	{attribute 'TcLinkTo' := '.bLimitForwardEnable:=TIIB[EL7041-1000_XRTM1_Ydwn]^STM Status^Status^Digital input 1;
                              .bLimitBackwardEnable:=TIIB[EL7041-1000_XRTM1_Ydwn]^STM Status^Status^Digital input 2'}
	{attribute 'pytmc' := '
		pv: XRTMR1:HOMS:MMS:YDWN
	'}
	M2 : DUT_MotionStage := (fVelocity:=200.0, nEnableMode:=ENUM_StageEnableMode.ALWAYS, bPowerSelf:=TRUE); // XRTM1 Ydwn
	fbMotionStage_m2 : FB_MotionStage;

	{attribute 'TcLinkTo' := '.bLimitForwardEnable:=TIIB[EL7041-1000_XRTM1_Xup]^STM Status^Status^Digital input 1;
                              .bLimitBackwardEnable:=TIIB[EL7041-1000_XRTM1_Xup]^STM Status^Status^Digital input 2'}
	{attribute 'pytmc' := '
		pv: XRTMR1:HOMS:MMS:XUP
	'}
	M3 : DUT_MotionStage := (fVelocity:=1000.0, nEnableMode:=ENUM_StageEnableMode.ALWAYS, bPowerSelf:=TRUE); // XRTM1 Xup
	fbMotionStage_m3 : FB_MotionStage;

	{attribute 'TcLinkTo' := '.bLimitForwardEnable:=TIIB[EL7041-1000_XRTM1_Xdwn]^STM Status^Status^Digital input 1;
                              .bLimitBackwardEnable:=TIIB[EL7041-1000_XRTM1_Xdwn]^STM Status^Status^Digital input 2'}
	{attribute 'pytmc' := '
		pv: XRTMR1:HOMS:MMS:XDWN
	'}
	M4 : DUT_MotionStage := (fVelocity:=1000.0, nEnableMode:=ENUM_StageEnableMode.ALWAYS, bPowerSelf:=TRUE); // XRTM1 Xdwn
	fbMotionStage_m4 : FB_MotionStage;

	{attribute 'TcLinkTo' := '.bLimitForwardEnable:=TIIB[EL7041-1000_XRTM1_PitchCoarse]^STM Status^Status^Digital input 1;
                              .bLimitBackwardEnable:=TIIB[EL7041-1000_XRTM1_PitchCoarse]^STM Status^Status^Digital input 2'}
	{attribute 'pytmc' := '
		pv: XRTMR1:HOMS:MMS:PITCH
	'}
	M5 : DUT_MotionStage := (fVelocity:=150.0); // XRTM1 Pitch Stepper

	{attribute 'TcLinkTo' := '.bLimitForwardEnable:=TIIB[EL7041-1000_XRTM1_Bender]^STM Status^Status^Digital input 1;
                              .bLimitBackwardEnable:=TIIB[EL7041-1000_XRTM1_Bender]^STM Status^Status^Digital input 2'}
	{attribute 'pytmc' := '
		pv: XRTMR1:HOMS:MMS:BENDER
	'}
	M6 : DUT_MotionStage := (fVelocity:=150.0, nEnableMode:=ENUM_StageEnableMode.ALWAYS, bPowerSelf:=TRUE); // XRTM1 Bender
	fbMotionStage_m6 : FB_MotionStage;

	{attribute 'TcLinkTo' := '.fbRunHOMS.bSTOEnable1:=TIIB[EL1004_XRTM1_STO]^Channel 1^Input;
                              .fbRunHOMS.bSTOEnable2:=TIIB[EL1004_XRTM1_STO]^Channel 2^Input;
	                          .fbRunHOMS.stYupEnc.Count:=TIIB[EL5042_XRTM1_Yupdwn]^FB Inputs Channel 1^Position;
	                          .fbRunHOMS.stYdwnEnc.Count:=TIIB[EL5042_XRTM1_Yupdwn]^FB Inputs Channel 2^Position;
	                          .fbRunHOMS.stXupEnc.Count:=TIIB[EL5042_XRTM1_Xupdwn]^FB Inputs Channel 1^Position;
	                          .fbRunHOMS.stXdwnEnc.Count:=TIIB[EL5042_XRTM1_Xupdwn]^FB Inputs Channel 2^Position'}
	{attribute 'pytmc' := '
		pv: XRTMR1:HOMS
	'}
	XRTM1 : DUT_HOMS;

	// Encoder Arrays/RMS Watch:
	{attribute 'pytmc' := '
		pv: XRTMR1:HOMS:ENC:Y
	'}
	fbYRMSErrorXRTM1 : FB_RMSWatch;
	fMaxYRMSErrorXRTM1 : LREAL;
	fMinYRMSErrorXRTM1 : LREAL;

	{attribute 'pytmc' := '
		pv: XRTMR1:HOMS:ENC:X
	'}
	fbXRMSErrorXRTM1 : FB_RMSWatch;
	fMaxXRMSErrorXRTM1 : LREAL;
	fMinXRMSErrorXRTM1 : LREAL;

	{attribute 'pytmc' := '
		pv: XRTMR1:HOMS:ENC:PITCH
	'}
	fbPitchRMSErrorXRTM1 : FB_RMSWatch;
	fMaxPitchRMSErrorXRTM1 : LREAL;
	fMinPitchRMSErrorXRTM1 : LREAL;

	{attribute 'pytmc' := '
		pv: XRTMR1:HOMS:ENC:BENDER
	'}
	fbBenderRMSErrorXRTM1 : FB_RMSWatch;
	fMaxBenderRMSErrorXRTM1 : LREAL;
	fMinBenderRMSErrorXRTM1 : LREAL;

	// Pitch Control
	fbXRTM1PitchControl : FB_PitchControl;
	bXRTM1PitchDone : BOOL;
	bXRTM1PitchBusy : BOOL;

	// Bender Control
	fbBenderXRTM1 : FB_Bender;

	// Raw Encoder Counts
	{attribute 'pytmc' := '
		pv: XRTMR1:HOMS:ENC:YUP:CNT
		field: EGU cnt
		io: i
	'}
	nEncCntYupXRTM1 : UDINT;
	{attribute 'pytmc' := '
		pv: XRTMR1:HOMS:ENC:YDWN:CNT
		field: EGU cnt
		io: i
	'}
	nEncCntYdwnXRTM1 : UDINT;
	{attribute 'pytmc' := '
		pv: XRTMR1:HOMS:ENC:XUP:CNT
		field: EGU cnt
		io: i
	'}
	nEncCntXupXRTM1 : UDINT;
	{attribute 'pytmc' := '
		pv: XRTMR1:HOMS:ENC:XDWN:CNT
		field: EGU cnt
		io: i
	'}
	nEncCntXdwnXRTM1 : UDINT;
	{attribute 'pytmc' := '
		pv: XRTMR1:HOMS:ENC:PITCH:CNT
		field: EGU cnt
		io: i
	'}
	nEncCntPitchXRTM1 : UDINT;

	// Encoder Reference Values
	{attribute 'pytmc' := '
		pv: XRTMR1:HOMS:ENC:YUP:REF
		field: EGU cnt
		io: i
	'}
	nEncRefYupXRTM1 : UDINT;
	{attribute 'pytmc' := '
		pv: XRTMR1:HOMS:ENC:YDWN:REF
		field: EGU cnt
		io: i
	'}
	nEncRefYdwnXRTM1 : UDINT;
	{attribute 'pytmc' := '
		pv: XRTMR1:HOMS:ENC:XUP:REF
		field: EGU cnt
		io: i
	'}
	nEncRefXupXRTM1 : UDINT;
	{attribute 'pytmc' := '
		pv: XRTMR1:HOMS:ENC:XDWN:REF
		field: EGU cnt
		io: i
	'}
	nEncRefXdwnXRTM1 : UDINT;
	{attribute 'pytmc' := '
		pv: XRTMR1:HOMS:ENC:PITCH:REF
		field: EGU cnt
		io: i
	'}
	nEncRefPitchXRTM1 : UDINT;
	mcReadParameterPitchXRTM1 : MC_ReadParameter;
	fEncRefPitchXRTM1_urad : LREAL; // Current Pitch encoder offset in urad
	
    //****** HOMS M2 and M3 **************************
	tpImAPLC : TP := (PT:=T#10S);
	ExpertMode	:	BOOL := FALSE;
	PitchManualMode: BOOL := FALSE;
	
	//Drive CoE Fb
	fbY1CoE	:	FB_ElmoGDCBellCoE;
	fbY2CoE	:	FB_ElmoGDCBellCoE;
	
	fbX1CoE	:	FB_ElmoGDCBellCoE;
	fbX2CoE	:	FB_ElmoGDCBellCoE;
	
	fbP1CoE	:	FB_ElmoGDCBellCoE;
	fbB1CoE	:	FB_ElmoGDCBellCoE;
	
	//Init params trigger
	rtInitParams	:	R_TRIG;
	
	//Test Parameters
	rStepSize: REAL;
	SettleTime: TON := (
	PT:=T#2s);
	TestUpperVoltage: REAL := 100;
	TestLowerVoltage: REAL := 10;
	xRunPiezoRepeatTest: BOOL;
	
	//Drive reference initializations
	fbInitDriveRef	:	FB_InitDriveRefs;
	//MPS Information
	fbMPS_States :  FB_MPS_STATES;
	M2_INRANGE  :   ARRAY[0..1] OF DINT := [24568920, 26568920];
	M2_OUTRANGE  :  ARRAY[0..1] OF DINT := [43568250, 50570250];
	//noConsequence	:	BOOL;
	
	mcBenderPower	:	MC_POWER;
	
	// HOMS M2
	XRTM2PitchControl	    :	FB_PitchControlOld;
	XRTM2Y_GantryControl	:	FB_Gantry;
	XRTM2X_GantryControl	:	FB_Gantry;
	
	fbM2Y1LS	:	FB_LimitSwitchState;
	fbM2Y2LS	:	FB_LimitSwitchState;
	fbM2X1LS	:	FB_LimitSwitchState;
	fbM2X2LS	:	FB_LimitSwitchState;
	fbM2P1LS	:	FB_PitchSoftLimits;	
	
    // HOMS M3
	XRTM3PitchControl	    :	FB_PitchControlOld;
	XRTM3Y_GantryControl	:	FB_Gantry;
	XRTM3X_GantryControl	:	FB_Gantry;
	
	fbM3Y1LS	:	FB_LimitSwitchState;
	fbM3Y2LS	:	FB_LimitSwitchState;
	fbM3X1LS	:	FB_LimitSwitchState;
	fbM3X2LS	:	FB_LimitSwitchState;
	fbM3P1LS	:	FB_PitchSoftLimits;	
	
	//************** **** *** ** *
	
	
	
	// PMPS arbiter interface
	fbArbiterIO : FB_SubSysToArbiter_IO;
	
	// Common
	fEncLeverArm_mm : LREAL := 513.0;
	// Logging
	fbLogHandler : FB_LogHandler;

END_VAR

// XRTM1
XRTM1.fbRunHOMS(stYup:=M1,
               stYdwn:=M2,
               stXup:=M3,
               stXdwn:=M4,
               stPitch:=M5,
	           nYupEncRef:=GVL_XRTM1_Constants.nYUP_ENC_REF,
               nYdwnEncRef:=GVL_XRTM1_Constants.nYDWN_ENC_REF,
               nXupEncRef:=GVL_XRTM1_Constants.nXUP_ENC_REF,
               nXdwnEncRef:=GVL_XRTM1_Constants.nXDWN_ENC_REF,
			   bExecuteCoupleY:=XRTM1.bExecuteCoupleY,
               bExecuteCoupleX:=XRTM1.bExecuteCoupleX,
			   bExecuteDecoupleY:=XRTM1.bExecuteDecoupleY,
               bExecuteDecoupleX:=XRTM1.bExecuteDecoupleX,
               bGantryAlreadyCoupledY=>XRTM1.bGantryAlreadyCoupledY,
               bGantryAlreadyCoupledX=>XRTM1.bGantryAlreadyCoupledX,
               nCurrGantryY=>XRTM1.nCurrGantryY,
               nCurrGantryX=>XRTM1.nCurrGantryX);
fbBenderXRTM1(stBender:=M6,
	         bSTOEnable1:=XRTM1.fbRunHOMS.bSTOEnable1,
		     bSTOEnable2:=XRTM1.fbRunHOMS.bSTOEnable2);
// No slave motion through Epics
M2.bExecute := FALSE; // XRTM1-Ydwn
M4.bExecute := FALSE; // XRTM1-Xdwn

// Convert nCurrGantry to um (smaller number) to read out in epics
XRTM1.fCurrGantryY_um := LINT_TO_REAL(XRTM1.nCurrGantryY) / 1000.0;
XRTM1.fCurrGantryX_um := LINT_TO_REAL(XRTM1.nCurrGantryX) / 1000.0;

// FB_MotionStage's for non-piezo axes
fbMotionStage_m1(stMotionStage:=M1);
fbMotionStage_m2(stMotionStage:=M2);
fbMotionStage_m3(stMotionStage:=M3);
fbMotionStage_m4(stMotionStage:=M4);
fbMotionStage_m6(stMotionStage:=M6);

// Calculate Pitch RMS Error:
fbYRMSErrorXRTM1(stMotionStage:=M1,
	            fMaxRMSError=>fMaxYRMSErrorXRTM1,
				fMinRMSError=>fMinYRMSErrorXRTM1);

fbXRMSErrorXRTM1(stMotionStage:=M3,
	            fMaxRMSError=>fMaxXRMSErrorXRTM1,
				fMinRMSError=>fMinXRMSErrorXRTM1);

fbPitchRMSErrorXRTM1(stMotionStage:=M5,
	                fMaxRMSError=>fMaxPitchRMSErrorXRTM1,
					fMinRMSError=>fMinPitchRMSErrorXRTM1);

fbBenderRMSErrorXRTM1(stMotionStage:=M6,
	                 fMaxRMSError=>fMaxBenderRMSErrorXRTM1,
					 fMinRMSError=>fMinBenderRMSErrorXRTM1);
// Pitch Control
fbXRTM1PitchControl(Pitch:=GVL_XRTM1.XRTM1_Pitch,
				   Stepper:=M5,
				   lrCurrentSetpoint:=M5.fPosition,
                   q_bDone=>bXRTM1PitchDone,
                   q_bBusy=>bXRTM1PitchBusy);
// When STO hit, need to reset SP
IF NOT M5.bHardwareEnable THEN
	M5.fPosition := M5.stAxisStatus.fActPosition;
END_IF

// Raw Encoder Counts For Epics
nEncCntYupXRTM1 := ULINT_TO_UDINT(XRTM1.fbRunHOMS.stYupEnc.Count);
nEncCntYdwnXRTM1 := ULINT_TO_UDINT(XRTM1.fbRunHOMS.stYdwnEnc.Count);
nEncCntXupXRTM1 := ULINT_TO_UDINT(XRTM1.fbRunHOMS.stXupEnc.Count);
nEncCntXdwnXRTM1 := ULINT_TO_UDINT(XRTM1.fbRunHOMS.stXdwnEnc.Count);
nEncCntPitchXRTM1 := LINT_TO_UDINT(GVL_XRTM1.XRTM1_Pitch.diEncCnt);

// Encoder Reference Values For Epics
nEncRefYupXRTM1 := ULINT_TO_UDINT(GVL_XRTM1_Constants.nYUP_ENC_REF);
nEncRefYdwnXRTM1 := ULINT_TO_UDINT(GVL_XRTM1_Constants.nYDWN_ENC_REF);
nEncRefXupXRTM1 := ULINT_TO_UDINT(GVL_XRTM1_Constants.nXUP_ENC_REF);
nEncRefXdwnXRTM1 := ULINT_TO_UDINT(GVL_XRTM1_Constants.nXDWN_ENC_REF);
mcReadParameterPitchXRTM1(Axis:=M5.Axis,
	                     Enable:=TRUE,
				         ParameterNumber:=MC_AxisParameter.AxisEncoderOffset,
				         ReadMode:=READMODE_CYCLIC,
				         Value=>fEncRefPitchXRTM1_urad);

nEncRefPitchXRTM1 := LREAL_TO_UDINT(ABS(fEncRefPitchXRTM1_urad) * fEncLeverArm_mm);

// HOMS ************************ ***** **** *** ** *
p_ModbusRx_OutputCoils();
p_ModbusRx_PLCMemory();

//InitParams
////////////////////
rtInitParams(CLK:=gFirstPass);
IF rtInitParams.Q THEN
	Init_XRTM2();
	Init_XRTM3();
	gFirstPass := FALSE;
END_IF

//System Error Handling
/////////////////////////////////////
//SystemErrorSummary(); //Check this action for a summary of all system faults
					  
//SystemError();

//Driver Parameter Verification
/////////////////////////////////////

//Gantry Interlock Logic
/////////////////////////////////////
	//SimGantry.VAxis.i_xMotorInterlock := TRUE;
	//SimGantry.PAxis.i_xMotorInterlock := TRUE;
	//SimGantry.SAxis.i_xMotorInterlock := TRUE;
	
LimitSwitchIO();

// Pitch control
/////////////////////////////////////
XRTM2PitchControl(Pitch:=HOMS2_Pitch, DirectPiezoMode:=(ExpertMode AND PitchManualMode), q_xDone=>HOMS2_Pitch.Axis.bDone, q_xBusy => HOMS2_Pitch.Axis.bBusy);
XRTM3PitchControl(Pitch:=HOMS3_Pitch, DirectPiezoMode:=(ExpertMode AND PitchManualMode), q_xDone=>HOMS3_Pitch.Axis.bDone, q_xBusy => HOMS3_Pitch.Axis.bBusy);
//Y motion
/////////////////////////////////////
HOMS3_YGantry.PAxis.stAxis.ReadStatus();
HOMS3_YGantry.SAxis.stAxis.ReadStatus();
HOMS3_YGantry.PAxis.stStatus.rActPosition := LREAL_TO_REAL(HOMS3_YGantry.PAxis.stAxis.NcToPlc.ActPos);
HOMS3_YGantry.SAxis.stStatus.rActPosition := LREAL_TO_REAL(HOMS3_YGantry.SAxis.stAxis.NcToPlc.ActPos);

//X Motion
/////////////////////////////////////
XRTM2X_GantryControl(Gantry:=HOMS2_XGantry);
XRTM3X_GantryControl(Gantry:=HOMS3_XGantry);

//Communicate state to MPS
////////////////////////////////
fbMPS_States(GANTRY:=HOMS2_XGantry,
			 OUT_LS:=NOT HOMS2_XGantry.PAxis.xHiLS OR NOT HOMS2_XGantry.SAxis.xLoLS,
			 IN_RANGE:=M2_INRANGE,
			 OUT_RANGE:=M2_OUTRANGE);
			 
bXRT_M2_IN  := fbMPS_States.IN;
bXRT_M2_OUT := fbMPS_States.OUT;
//EPICS Tx Update
////////////////////
p_ModbusTx_InputCoils();
//p_ModbusTx_OutputCoils();
p_ModbusTx_InputReg();
p_ModbusTx_PLCMemory();

// **************************** ***** **** *** ** * HOMS


P_CoatingProtections();

// Logging
fbLogHandler();

// PMPS
GVL_PMPS.g_fbArbiter1.AddRequest(16#5, PMPS_GVL.cstFullBeam);
fbArbiterIO(Arbiter := GVL_PMPS.g_fbArbiter1, fbFFHWO := GVL_PMPS.g_FastFaultOutput1);
GVL_PMPS.g_FastFaultOutput1.Execute(i_xVeto:=);
GVL_PMPS.g_FastFaultOutput2.Execute(i_xVeto:=);

ACTION Init_XRTM2:
//FEE-M2
///////////////////////////


//Initialize ELMO Drive references
fbInitDriveRef(stCoE:=HOMS2_XGantry.PAxis.stCoE);
fbInitDriveRef(stCoE:=HOMS2_XGantry.SAxis.stCoE);
fbInitDriveRef(stCoE:=HOMS2_YGantry.PAxis.stCoE);
fbInitDriveRef(stCoE:=HOMS2_YGantry.SAxis.stCoE);
fbInitDriveRef(stCoE:=HOMS2_Pitch.Stepper.stCoE);

//Initialze Drive Speeds and Accelerations
//////////////////////////////////////////
HOMS2_XGantry.PAxis.fAcceleration := 1.0;
HOMS2_XGantry.SAxis.fAcceleration := 1.0;
HOMS2_YGantry.PAxis.fAcceleration := 1.0;
HOMS2_YGantry.SAxis.fAcceleration := 1.0;

HOMS2_XGantry.PAxis.fDeceleration := 1.0;
HOMS2_XGantry.SAxis.fDeceleration := 1.0;
HOMS2_YGantry.PAxis.fDeceleration := 1.0;
HOMS2_YGantry.SAxis.fDeceleration := 1.0;

HOMS2_XGantry.PAxis.fVelocity := 0.1;
HOMS2_XGantry.SAxis.fVelocity := 0.1;
HOMS2_YGantry.PAxis.fVelocity := 0.1;
HOMS2_YGantry.SAxis.fVelocity := 0.1;

HOMS2_Pitch.Stepper.fAcceleration := 39;
HOMS2_Pitch.Stepper.fDeceleration := 39;
HOMS2_Pitch.Stepper.fVelocity     := 100;

//Initialize Piezo Driver
/////////////////////////////////////
HOMS2_Pitch.Piezo.stPIParams.fKp := 0.001;
HOMS2_Pitch.Piezo.stPIParams.tTn := T#500MS;
HOMS2_Pitch.Piezo.stPIParams.fOutMaxLimit := 1;
HOMS2_Pitch.Piezo.stPIParams.fOutMinLimit := -1;
END_ACTION

ACTION Init_XRTM3:
//FEE-M3
///////////////////////////


//Initialize ELMO Drive references
fbInitDriveRef(stCoE:=HOMS3_XGantry.PAxis.stCoE);
fbInitDriveRef(stCoE:=HOMS3_XGantry.SAxis.stCoE);
fbInitDriveRef(stCoE:=HOMS3_YGantry.PAxis.stCoE);
fbInitDriveRef(stCoE:=HOMS3_YGantry.SAxis.stCoE);
fbInitDriveRef(stCoE:=HOMS3_Pitch.Stepper.stCoE);

//Initialze Drive Speeds and Accelerations
//////////////////////////////////////////
HOMS3_XGantry.PAxis.fAcceleration := 1.0;
HOMS3_XGantry.SAxis.fAcceleration := 1.0;
HOMS3_YGantry.PAxis.fAcceleration := 1.0;
HOMS3_YGantry.SAxis.fAcceleration := 1.0;

HOMS3_XGantry.PAxis.fDeceleration := 1.0;
HOMS3_XGantry.SAxis.fDeceleration := 1.0;
HOMS3_YGantry.PAxis.fDeceleration := 1.0;
HOMS3_YGantry.SAxis.fDeceleration := 1.0;

HOMS3_XGantry.PAxis.fVelocity := 0.1;
HOMS3_XGantry.SAxis.fVelocity := 0.1;
HOMS3_YGantry.PAxis.fVelocity := 0.1;
HOMS3_YGantry.SAxis.fVelocity := 0.1;

HOMS3_Pitch.Stepper.fAcceleration := 39;
HOMS3_Pitch.Stepper.fDeceleration := 39;
HOMS3_Pitch.Stepper.fVelocity     := 100;

//Initialize Piezo Driver
/////////////////////////////////////
HOMS3_Pitch.Piezo.stPIParams.fKp := 0.001;
HOMS3_Pitch.Piezo.stPIParams.tTn := T#500MS;
HOMS3_Pitch.Piezo.stPIParams.fOutMaxLimit := 1;
HOMS3_Pitch.Piezo.stPIParams.fOutMinLimit := -1;
END_ACTION

ACTION LimitSwitchIO:
//XRT M2
//////////////////////////
fbM2Y1LS(diInputs:=HOMS2_YGantry.PAxis.diInputs, 
xHiLS=>HOMS2_YGantry.PAxis.xHiLS,
xLoLS=>HOMS2_YGantry.PAxis.xLoLS,
STO => gM2STO);

fbM2Y2LS(diInputs:=HOMS2_YGantry.SAxis.diInputs, 
xHiLS=>HOMS2_YGantry.SAxis.xHiLS,
xLoLS=>HOMS2_YGantry.SAxis.xLoLS);

fbM2X1LS(diInputs:=HOMS2_XGantry.PAxis.diInputs, 
xHiLS=>HOMS2_XGantry.PAxis.xHiLS,
xLoLS=>HOMS2_XGantry.PAxis.xLoLS);

fbM2X2LS(diInputs:=HOMS2_XGantry.SAxis.diInputs, 
xHiLS=>HOMS2_XGantry.SAxis.xHiLS,
xLoLS=>HOMS2_XGantry.SAxis.xLoLS);

fbM2P1LS(Pitch:=HOMS2_Pitch,
xHiLS=>HOMS2_Pitch.Stepper.xHiLS,
xLoLS=>HOMS2_Pitch.Stepper.xLoLS);

//XRT M3
//////////////////////////
fbM3Y1LS(diInputs:=HOMS3_YGantry.PAxis.diInputs, 
xHiLS=>HOMS3_YGantry.PAxis.xHiLS,
xLoLS=>HOMS3_YGantry.PAxis.xLoLS,
STO => gM3STO);

fbM3Y2LS(diInputs:=HOMS3_YGantry.SAxis.diInputs, 
xHiLS=>HOMS3_YGantry.SAxis.xHiLS,
xLoLS=>HOMS3_YGantry.SAxis.xLoLS);

fbM3X1LS(diInputs:=HOMS3_XGantry.PAxis.diInputs, 
xHiLS=>HOMS3_XGantry.PAxis.xHiLS,
xLoLS=>HOMS3_XGantry.PAxis.xLoLS);
(*
fbM3X2LS(diInputs:=HOMS3_XGantry.PAxis.diInputs,  //Paxis is here on purpose <HACK>
xHiLS=>HOMS3_XGantry.SAxis.xHiLS,
xLoLS=>HOMS3_XGantry.SAxis.xLoLS);
*)
fbM3X2LS(diInputs:=HOMS3_XGantry.SAxis.diInputs,  // Switching to SAxis works as expected, reason for <HACK> unclear
xHiLS=>HOMS3_XGantry.SAxis.xHiLS,
xLoLS=>HOMS3_XGantry.SAxis.xLoLS);

fbM3P1LS(Pitch:=HOMS3_Pitch,
xHiLS=>HOMS3_Pitch.Stepper.xHiLS,
xLoLS=>HOMS3_Pitch.Stepper.xLoLS);
END_ACTION

END_PROGRAM

// ---- POUs/Modbus/p_ModbusRx_OutputCoils.TcPOU
PROGRAM p_ModbusRx_OutputCoils
VAR
	
END_VAR

HOMS2_XGantry.PAxis.bTwkFwd:=mb_Output_Coils[60];
HOMS2_XGantry.PAxis.bTwkBwd:=mb_Output_Coils[61];
HOMS2_XGantry.SAxis.bTwkFwd:=mb_Output_Coils[62];
HOMS2_XGantry.SAxis.bTwkBwd:=mb_Output_Coils[63];
HOMS2_YGantry.PAxis.bTwkFwd:=mb_Output_Coils[64];
HOMS2_YGantry.PAxis.bTwkBwd:=mb_Output_Coils[65];
HOMS2_YGantry.SAxis.bTwkFwd:=mb_Output_Coils[66];
HOMS2_YGantry.SAxis.bTwkBwd:=mb_Output_Coils[67];
HOMS2_Pitch.Axis.bTwkFwd:=mb_Output_Coils[68];
HOMS2_Pitch.Axis.bTwkBwd:=mb_Output_Coils[69];
HOMS2_Pitch.Axis.xStop:=mb_Output_Coils[73];
HOMS2_XGantry.xUncouple:=mb_Output_Coils[76];
HOMS2_YGantry.xUncouple:=mb_Output_Coils[77];
HOMS3_XGantry.PAxis.bTwkFwd:=mb_Output_Coils[78];
HOMS3_XGantry.PAxis.bTwkBwd:=mb_Output_Coils[79];
HOMS3_XGantry.SAxis.bTwkFwd:=mb_Output_Coils[80];
HOMS3_XGantry.SAxis.bTwkBwd:=mb_Output_Coils[81];
HOMS3_YGantry.PAxis.bTwkFwd:=mb_Output_Coils[82];
HOMS3_YGantry.PAxis.bTwkBwd:=mb_Output_Coils[83];
HOMS3_YGantry.SAxis.bTwkFwd:=mb_Output_Coils[84];
HOMS3_YGantry.SAxis.bTwkBwd:=mb_Output_Coils[85];
HOMS3_Pitch.Axis.bTwkFwd:=mb_Output_Coils[86];
HOMS3_Pitch.Axis.bTwkBwd:=mb_Output_Coils[87];
HOMS3_Pitch.Piezo.xEnable:=mb_Output_Coils[88];
HOMS3_Pitch.Axis.xStop:=mb_Output_Coils[89];
HOMS3_XGantry.xUncouple:=mb_Output_Coils[90];
HOMS3_YGantry.xUncouple:=mb_Output_Coils[91];
HOMS2_XGantry.PAxis.xReset := mb_Output_Coils[95];
HOMS2_YGantry.PAxis.xReset := mb_Output_Coils[96];
HOMS2_Pitch.Axis.xReset := mb_Output_Coils[97];
HOMS3_XGantry.PAxis.xReset := mb_Output_Coils[98];
HOMS3_YGantry.PAxis.xReset := mb_Output_Coils[99];
HOMS3_Pitch.Axis.xReset := mb_Output_Coils[100];

END_PROGRAM

// ---- POUs/Modbus/p_ModbusRx_PLCMemory.TcPOU
PROGRAM p_ModbusRx_PLCMemory
VAR
END_VAR

MEMCPY(srcAddr:=ADR(mb_PLC_Memory[20]), destAddr:=ADR(HOMS2_XGantry.PAxis.rReqAbsolute), n:=SIZEOF(HOMS2_XGantry.PAxis.rReqAbsolute));
MEMCPY(srcAddr:=ADR(mb_PLC_Memory[22]), destAddr:=ADR(HOMS2_XGantry.PAxis.rTweak), n:=SIZEOF(HOMS2_XGantry.PAxis.rTweak));
MEMCPY(srcAddr:=ADR(mb_PLC_Memory[24]), destAddr:=ADR(HOMS2_XGantry.SAxis.rReqAbsolute), n:=SIZEOF(HOMS2_XGantry.SAxis.rReqAbsolute));
MEMCPY(srcAddr:=ADR(mb_PLC_Memory[26]), destAddr:=ADR(HOMS2_XGantry.SAxis.rTweak), n:=SIZEOF(HOMS2_XGantry.SAxis.rTweak));
MEMCPY(srcAddr:=ADR(mb_PLC_Memory[28]), destAddr:=ADR(HOMS2_YGantry.PAxis.rReqAbsolute), n:=SIZEOF(HOMS2_YGantry.PAxis.rReqAbsolute));
MEMCPY(srcAddr:=ADR(mb_PLC_Memory[30]), destAddr:=ADR(HOMS2_YGantry.PAxis.rTweak), n:=SIZEOF(HOMS2_YGantry.PAxis.rTweak));
MEMCPY(srcAddr:=ADR(mb_PLC_Memory[32]), destAddr:=ADR(HOMS2_YGantry.SAxis.rReqAbsolute), n:=SIZEOF(HOMS2_YGantry.SAxis.rReqAbsolute));
MEMCPY(srcAddr:=ADR(mb_PLC_Memory[34]), destAddr:=ADR(HOMS2_YGantry.SAxis.rTweak), n:=SIZEOF(HOMS2_YGantry.SAxis.rTweak));
MEMCPY(srcAddr:=ADR(mb_PLC_Memory[36]), destAddr:=ADR(HOMS2_Pitch.Axis.rReqAbsPos), n:=SIZEOF(HOMS2_Pitch.Axis.rReqAbsPos));
MEMCPY(srcAddr:=ADR(mb_PLC_Memory[38]), destAddr:=ADR(HOMS2_Pitch.Axis.rTweak), n:=SIZEOF(HOMS2_Pitch.Axis.rTweak));
MEMCPY(srcAddr:=ADR(mb_PLC_Memory[40]), destAddr:=ADR(HOMS3_XGantry.PAxis.rReqAbsolute), n:=SIZEOF(HOMS3_XGantry.PAxis.rReqAbsolute));
MEMCPY(srcAddr:=ADR(mb_PLC_Memory[42]), destAddr:=ADR(HOMS3_XGantry.PAxis.rTweak), n:=SIZEOF(HOMS3_XGantry.PAxis.rTweak));
MEMCPY(srcAddr:=ADR(mb_PLC_Memory[44]), destAddr:=ADR(HOMS3_XGantry.SAxis.rReqAbsolute), n:=SIZEOF(HOMS3_XGantry.SAxis.rReqAbsolute));
MEMCPY(srcAddr:=ADR(mb_PLC_Memory[46]), destAddr:=ADR(HOMS3_XGantry.SAxis.rTweak), n:=SIZEOF(HOMS3_XGantry.SAxis.rTweak));
MEMCPY(srcAddr:=ADR(mb_PLC_Memory[48]), destAddr:=ADR(HOMS3_YGantry.PAxis.rReqAbsolute), n:=SIZEOF(HOMS3_YGantry.PAxis.rReqAbsolute));
MEMCPY(srcAddr:=ADR(mb_PLC_Memory[50]), destAddr:=ADR(HOMS3_YGantry.PAxis.rTweak), n:=SIZEOF(HOMS3_YGantry.PAxis.rTweak));
MEMCPY(srcAddr:=ADR(mb_PLC_Memory[52]), destAddr:=ADR(HOMS3_YGantry.SAxis.rReqAbsolute), n:=SIZEOF(HOMS3_YGantry.SAxis.rReqAbsolute));
MEMCPY(srcAddr:=ADR(mb_PLC_Memory[54]), destAddr:=ADR(HOMS3_YGantry.SAxis.rTweak), n:=SIZEOF(HOMS3_YGantry.SAxis.rTweak));
MEMCPY(srcAddr:=ADR(mb_PLC_Memory[56]), destAddr:=ADR(HOMS3_Pitch.Axis.rReqAbsPos), n:=SIZEOF(HOMS3_Pitch.Axis.rReqAbsPos));
MEMCPY(srcAddr:=ADR(mb_PLC_Memory[58]), destAddr:=ADR(HOMS3_Pitch.Axis.rTweak), n:=SIZEOF(HOMS3_Pitch.Stepper.rTweak));

MEMCPY(srcAddr:=ADR(mb_PLC_Memory[64]), destAddr:=ADR(HOMS2_Pitch.Stepper.rStepperDmovRange), n:=SIZEOF(HOMS2_Pitch.Stepper.rStepperDmovRange));
MEMCPY(srcAddr:=ADR(mb_PLC_Memory[66]), destAddr:=ADR(HOMS2_Pitch.Piezo.rPiezoDmovRange), n:=SIZEOF(HOMS2_Pitch.Piezo.rPiezoDmovRange));
MEMCPY(srcAddr:=ADR(mb_PLC_Memory[68]), destAddr:=ADR(HOMS3_Pitch.Stepper.rStepperDmovRange), n:=SIZEOF(HOMS3_Pitch.Stepper.rStepperDmovRange));
MEMCPY(srcAddr:=ADR(mb_PLC_Memory[70]), destAddr:=ADR(HOMS3_Pitch.Piezo.rPiezoDmovRange), n:=SIZEOF(HOMS3_Pitch.Piezo.rPiezoDmovRange));

//MEMCPY(srcAddr:=ADR(mb_PLC_Memory[140]), destAddr:=ADR(HOMS1_Pitch.Piezo.rReqVoltage), n:=SIZEOF(HOMS1_Pitch.Piezo.rReqVoltage));
//MEMCPY(srcAddr:=ADR(mb_PLC_Memory[142]), destAddr:=ADR(HOMS2_Pitch.Piezo.rReqVoltage), n:=SIZEOF(HOMS2_Pitch.Piezo.rReqVoltage));

END_PROGRAM

// ---- POUs/Modbus/p_ModbusTx_InputCoils.TcPOU
PROGRAM p_ModbusTx_InputCoils
VAR

END_VAR

VAR_OUTPUT

END_VAR

mb_Input_Coils[30]:=HOMS2_XGantry.PAxis.stAxis.Status.StandStill;
mb_Input_Coils[31]:=HOMS2_XGantry.PAxis.bDone;
mb_Input_Coils[32]:=HOMS2_XGantry.PAxis.xHiLS;
mb_Input_Coils[33]:=HOMS2_XGantry.PAxis.xLoLS;
mb_Input_Coils[34]:=HOMS2_XGantry.PAxis.i_xMotorInterlock;
mb_Input_Coils[35]:=HOMS2_XGantry.PAxis.xEnable ;
mb_Input_Coils[36]:=HOMS2_XGantry.SAxis.stAxis.Status.StandStill;
mb_Input_Coils[37]:=HOMS2_XGantry.SAxis.bDone;
mb_Input_Coils[38]:=HOMS2_XGantry.SAxis.xHiLS;
mb_Input_Coils[39]:=HOMS2_XGantry.SAxis.xLoLS;
mb_Input_Coils[40]:=HOMS2_XGantry.SAxis.i_xMotorInterlock;
mb_Input_Coils[41]:=HOMS2_XGantry.SAxis.xEnable ;
mb_Input_Coils[42]:=HOMS2_YGantry.PAxis.stAxis.Status.StandStill;
mb_Input_Coils[43]:=HOMS2_YGantry.PAxis.bDone;
mb_Input_Coils[44]:=HOMS2_YGantry.PAxis.xHiLS;
mb_Input_Coils[45]:=HOMS2_YGantry.PAxis.xLoLS;
mb_Input_Coils[46]:=HOMS2_YGantry.PAxis.i_xMotorInterlock;
mb_Input_Coils[47]:=HOMS2_YGantry.PAxis.xEnable ;
mb_Input_Coils[48]:=HOMS2_YGantry.SAxis.stAxis.Status.StandStill;
mb_Input_Coils[49]:=HOMS2_YGantry.SAxis.bDone;
mb_Input_Coils[50]:=HOMS2_YGantry.SAxis.xHiLS;
mb_Input_Coils[51]:=HOMS2_YGantry.SAxis.xLoLS;
mb_Input_Coils[52]:=HOMS2_YGantry.SAxis.i_xMotorInterlock;
mb_Input_Coils[53]:=HOMS2_YGantry.SAxis.xEnable ;
mb_Input_Coils[54]:=HOMS2_Pitch.Axis.bBusy;
mb_Input_Coils[55]:=HOMS2_Pitch.Axis.bDone;
mb_Input_Coils[56]:=HOMS2_Pitch.Stepper.xHiLS;
mb_Input_Coils[57]:=HOMS2_Pitch.Stepper.xLoLS;
mb_Input_Coils[58]:=HOMS2_Pitch.Stepper.i_xMotorInterlock;
mb_Input_Coils[59]:=HOMS2_Pitch.Stepper.xEnable ;

mb_Input_Coils[68]:=HOMS2_XGantry.DiffFlt;
mb_Input_Coils[69]:=HOMS2_XGantry.vAxis.xHiLS;
mb_Input_Coils[70]:=HOMS2_XGantry.vAxis.xLoLS;
mb_Input_Coils[71]:=HOMS2_XGantry.VAxis.xEnable;
mb_Input_Coils[72]:=HOMS2_YGantry.DiffFlt;
mb_Input_Coils[73]:=HOMS2_YGantry.vAxis.xHiLS;
mb_Input_Coils[74]:=HOMS2_YGantry.vAxis.xLoLS;
mb_Input_Coils[75]:=HOMS2_YGantry.VAxis.xEnable;

mb_Input_Coils[77]:=NOT HOMS2_Pitch.Piezo.xIdleMode;
mb_Input_Coils[78]:=HOMS3_XGantry.PAxis.stAxis.Status.StandStill;
mb_Input_Coils[79]:=HOMS3_XGantry.PAxis.bDone;
mb_Input_Coils[80]:=HOMS3_XGantry.PAxis.xHiLS;
mb_Input_Coils[81]:=HOMS3_XGantry.PAxis.xLoLS;
mb_Input_Coils[82]:=HOMS3_XGantry.PAxis.i_xMotorInterlock;
mb_Input_Coils[83]:=HOMS3_XGantry.PAxis.xEnable ;
mb_Input_Coils[84]:=HOMS3_XGantry.SAxis.stAxis.Status.StandStill;
mb_Input_Coils[85]:=HOMS3_XGantry.SAxis.bDone;
mb_Input_Coils[86]:=HOMS3_XGantry.SAxis.xHiLS;
mb_Input_Coils[87]:=HOMS3_XGantry.SAxis.xLoLS;
mb_Input_Coils[88]:=HOMS3_XGantry.SAxis.i_xMotorInterlock;
mb_Input_Coils[89]:=HOMS3_XGantry.SAxis.xEnable ;
mb_Input_Coils[90]:=HOMS3_YGantry.PAxis.stAxis.Status.StandStill;
mb_Input_Coils[91]:=HOMS3_YGantry.PAxis.bDone;
mb_Input_Coils[92]:=HOMS3_YGantry.PAxis.xHiLS;
mb_Input_Coils[93]:=HOMS3_YGantry.PAxis.xLoLS;
mb_Input_Coils[94]:=HOMS3_YGantry.PAxis.i_xMotorInterlock;
mb_Input_Coils[95]:=HOMS3_YGantry.PAxis.xEnable ;
mb_Input_Coils[96]:=HOMS3_YGantry.SAxis.stAxis.Status.StandStill;
mb_Input_Coils[97]:=HOMS3_YGantry.SAxis.bDone;
mb_Input_Coils[98]:=HOMS3_YGantry.SAxis.xHiLS;
mb_Input_Coils[99]:=HOMS3_YGantry.SAxis.xLoLS;
mb_Input_Coils[100]:=HOMS3_YGantry.SAxis.i_xMotorInterlock;
mb_Input_Coils[101]:=HOMS3_YGantry.SAxis.xEnable ;
mb_Input_Coils[102]:=HOMS3_Pitch.Axis.bBusy;
mb_Input_Coils[103]:=HOMS3_Pitch.Axis.bDone;
mb_Input_Coils[104]:=HOMS3_Pitch.Stepper.xHiLS;
mb_Input_Coils[105]:=HOMS3_Pitch.Stepper.xLoLS;
mb_Input_Coils[106]:=HOMS3_Pitch.Stepper.i_xMotorInterlock;
mb_Input_Coils[107]:=HOMS3_Pitch.Stepper.xEnable ;
mb_Input_Coils[108]:=HOMS3_XGantry.DiffFlt;
mb_Input_Coils[109]:=HOMS3_XGantry.vAxis.xHiLS;
mb_Input_Coils[110]:=HOMS3_XGantry.vAxis.xLoLS;
mb_Input_Coils[111]:=HOMS3_XGantry.VAxis.xEnable;
mb_Input_Coils[112]:=HOMS3_YGantry.DiffFlt;
mb_Input_Coils[113]:=HOMS3_YGantry.vAxis.xHiLS;
mb_Input_Coils[114]:=HOMS3_YGantry.vAxis.xLoLS;
mb_Input_Coils[115]:=HOMS3_YGantry.VAxis.xEnable;
mb_Input_Coils[116]:=NOT HOMS3_Pitch.Piezo.xIdleMode;

mb_Input_Coils[119]:=HOMS2_XGantry.xCoupled;
mb_Input_Coils[120]:=HOMS2_YGantry.xCoupled;
mb_Input_Coils[121]:=HOMS3_XGantry.xCoupled;
mb_Input_Coils[122]:=HOMS3_YGantry.xCoupled;

END_PROGRAM

// ---- POUs/Modbus/p_ModbusTx_InputReg.TcPOU
PROGRAM p_ModbusTx_InputReg
VAR
	
END_VAR

mb_Input_Registers[0]:=0;  //System info
mb_Input_Registers[1]:=0;  //System info
mb_Input_Registers[2]:=0;  //System info
mb_Input_Registers[3]:=0;  //System info
mb_Input_Registers[4]:=0;  //System info
mb_Input_Registers[5]:=0;  //System info
mb_Input_Registers[6]:=0;  //System info
mb_Input_Registers[7]:=0;  //System info
mb_Input_Registers[8]:=0;  //System info
mb_Input_Registers[9]:=0;  //System info
mb_Input_Registers[10]:=0;  //VG pressure readbacks
mb_Input_Registers[11]:=0;  //VG pressure readbacks
mb_Input_Registers[12]:=0;  //VG pressure readbacks
mb_Input_Registers[13]:=0;  //VG pressure readbacks
mb_Input_Registers[14]:=0;  //VG pressure readbacks
mb_Input_Registers[15]:=0;  //VG pressure readbacks
mb_Input_Registers[16]:=0;  //VG pressure readbacks
mb_Input_Registers[17]:=0;  //VG pressure readbacks
mb_Input_Registers[18]:=0;  //VG pressure readbacks
mb_Input_Registers[19]:=0;  //VG pressure readbacks
mb_Input_Registers[20]:=0;  //VG pressure readbacks
mb_Input_Registers[21]:=0;  //VG pressure readbacks
mb_Input_Registers[22]:=0;  //VG pressure readbacks
mb_Input_Registers[23]:=0;  //VG pressure readbacks
mb_Input_Registers[24]:=0;  //VG pressure readbacks
mb_Input_Registers[25]:=0;  //VG pressure readbacks
mb_Input_Registers[26]:=0;  //VG pressure readbacks
mb_Input_Registers[27]:=0;  //VG pressure readbacks
mb_Input_Registers[28]:=0;  //VG pressure readbacks
mb_Input_Registers[29]:=0;  //VG pressure readbacks
mb_Input_Registers[30]:=0;  //VG pressure readbacks
mb_Input_Registers[31]:=0;  //VG pressure readbacks
mb_Input_Registers[32]:=0;  //VG pressure readbacks
mb_Input_Registers[33]:=0;  //VG pressure readbacks
mb_Input_Registers[34]:=0;  //VG pressure readbacks
mb_Input_Registers[35]:=0;  //VG pressure readbacks
mb_Input_Registers[36]:=0;  //VG pressure readbacks
mb_Input_Registers[37]:=0;  //VG pressure readbacks
mb_Input_Registers[38]:=0;  //VG pressure readbacks
mb_Input_Registers[39]:=0;  //VG pressure readbacks
mb_Input_Registers[40]:=0;  //VG pressure readbacks
mb_Input_Registers[41]:=0;  //VG pressure readbacks
mb_Input_Registers[42]:=0;  //VG pressure readbacks
mb_Input_Registers[43]:=0;  //VG pressure readbacks
mb_Input_Registers[44]:=0;  //VG pressure readbacks
mb_Input_Registers[45]:=0;  //VG pressure readbacks
mb_Input_Registers[46]:=0;  //VG pressure readbacks
mb_Input_Registers[47]:=0;  //VG pressure readbacks
mb_Input_Registers[48]:=0;  //VG pressure readbacks
mb_Input_Registers[49]:=0;  //VG pressure readbacks
mb_Input_Registers[50]:=0;  //VG pressure readbacks
mb_Input_Registers[51]:=0;  //VG pressure readbacks
mb_Input_Registers[52]:=0;  //VG pressure readbacks
mb_Input_Registers[53]:=0;  //VG pressure readbacks
mb_Input_Registers[54]:=0;  //VG pressure readbacks
mb_Input_Registers[55]:=0;  //VG pressure readbacks
mb_Input_Registers[56]:=0;  //VG pressure readbacks
mb_Input_Registers[57]:=0;  //VG pressure readbacks
mb_Input_Registers[58]:=0;  //VG pressure readbacks
mb_Input_Registers[59]:=0;  //VG pressure readbacks
mb_Input_Registers[60]:=0;  //VG pressure readbacks
mb_Input_Registers[61]:=0;  //VG pressure readbacks
mb_Input_Registers[62]:=0;  //VG pressure readbacks
mb_Input_Registers[63]:=0;  //VG pressure readbacks
mb_Input_Registers[64]:=0;  //VG pressure readbacks
mb_Input_Registers[65]:=0;  //VG pressure readbacks
mb_Input_Registers[66]:=0;  //VG pressure readbacks
mb_Input_Registers[67]:=0;  //VG pressure readbacks
mb_Input_Registers[68]:=0;  //VG pressure readbacks
mb_Input_Registers[69]:=0;  //VG pressure readbacks
mb_Input_Registers[70]:=0;  //VG state readbacks
mb_Input_Registers[71]:=0;  //VG state readbacks
mb_Input_Registers[72]:=0;  //VG state readbacks
mb_Input_Registers[73]:=0;  //VG state readbacks
mb_Input_Registers[74]:=0;  //VG state readbacks
mb_Input_Registers[75]:=0;  //VG state readbacks
mb_Input_Registers[76]:=0;  //VG state readbacks
mb_Input_Registers[77]:=0;  //VG state readbacks
mb_Input_Registers[78]:=0;  //VG state readbacks
mb_Input_Registers[79]:=0;  //VG state readbacks
mb_Input_Registers[80]:=0;  //VG state readbacks
mb_Input_Registers[81]:=0;  //VG state readbacks
mb_Input_Registers[82]:=0;  //VG state readbacks
mb_Input_Registers[83]:=0;  //VG state readbacks
mb_Input_Registers[84]:=0;  //VG state readbacks
mb_Input_Registers[85]:=0;  //VG state readbacks
mb_Input_Registers[86]:=0;  //VG state readbacks
mb_Input_Registers[87]:=0;  //VG state readbacks
mb_Input_Registers[88]:=0;  //VG state readbacks
mb_Input_Registers[89]:=0;  //VG state readbacks
mb_Input_Registers[90]:=0;  //VG state readbacks
mb_Input_Registers[91]:=0;  //VG state readbacks
mb_Input_Registers[92]:=0;  //VG state readbacks
mb_Input_Registers[93]:=0;  //VG state readbacks
mb_Input_Registers[94]:=0;  //VG state readbacks
mb_Input_Registers[95]:=0;  //VG state readbacks
mb_Input_Registers[96]:=0;  //VG state readbacks
mb_Input_Registers[97]:=0;  //VG state readbacks
mb_Input_Registers[98]:=0;  //VG state readbacks
mb_Input_Registers[99]:=0;  //VG state readbacks
mb_Input_Registers[100]:=0;  //VG state readbacks
mb_Input_Registers[101]:=0;  //VG state readbacks
mb_Input_Registers[102]:=0;  //VG state readbacks
mb_Input_Registers[103]:=0;  //VG state readbacks
mb_Input_Registers[104]:=0;  //VG state readbacks
mb_Input_Registers[105]:=0;  //VG state readbacks
mb_Input_Registers[106]:=0;  //VG state readbacks
mb_Input_Registers[107]:=0;  //VG state readbacks
mb_Input_Registers[108]:=0;  //VG state readbacks
mb_Input_Registers[109]:=0;  //VG state readbacks
mb_Input_Registers[110]:=0;  //VG state readbacks
mb_Input_Registers[111]:=0;  //VG state readbacks
mb_Input_Registers[112]:=0;  //VG state readbacks
mb_Input_Registers[113]:=0;  //VG state readbacks
mb_Input_Registers[114]:=0;  //VG state readbacks
mb_Input_Registers[115]:=0;  //VG state readbacks
mb_Input_Registers[116]:=0;  //VG state readbacks
mb_Input_Registers[117]:=0;  //VG state readbacks
mb_Input_Registers[118]:=0;  //VG state readbacks
mb_Input_Registers[119]:=0;  //VG state readbacks
mb_Input_Registers[120]:=0;  //default
mb_Input_Registers[121]:=0;  //default
mb_Input_Registers[122]:=0;  //default
mb_Input_Registers[123]:=0;  //default
mb_Input_Registers[124]:=0;  //default
mb_Input_Registers[125]:=0;  //default
mb_Input_Registers[126]:=0;  //default
mb_Input_Registers[127]:=0;  //default
mb_Input_Registers[128]:=0;  //default
mb_Input_Registers[129]:=0;  //default
mb_Input_Registers[130]:=0;  //default
mb_Input_Registers[131]:=0;  //default
mb_Input_Registers[132]:=0;  //default
mb_Input_Registers[133]:=0;  //default
mb_Input_Registers[134]:=0;  //default
mb_Input_Registers[135]:=0;  //default
mb_Input_Registers[136]:=0;  //default
mb_Input_Registers[137]:=0;  //default
mb_Input_Registers[138]:=0;  //default
mb_Input_Registers[139]:=0;  //default
mb_Input_Registers[140]:=0;  //default
mb_Input_Registers[141]:=0;  //default
mb_Input_Registers[142]:=0;  //default
mb_Input_Registers[143]:=0;  //default
mb_Input_Registers[144]:=0;  //default
mb_Input_Registers[145]:=0;  //default
mb_Input_Registers[146]:=0;  //default
mb_Input_Registers[147]:=0;  //default
mb_Input_Registers[148]:=0;  //default
mb_Input_Registers[149]:=0;  //default
mb_Input_Registers[150]:=0;  //default
mb_Input_Registers[151]:=0;  //default
mb_Input_Registers[152]:=0;  //default
mb_Input_Registers[153]:=0;  //default
mb_Input_Registers[154]:=0;  //default
mb_Input_Registers[155]:=0;  //default
mb_Input_Registers[156]:=0;  //default
mb_Input_Registers[157]:=0;  //default
mb_Input_Registers[158]:=0;  //default
mb_Input_Registers[159]:=0;  //default
mb_Input_Registers[160]:=0;  //default
mb_Input_Registers[161]:=0;  //default
mb_Input_Registers[162]:=0;  //default
mb_Input_Registers[163]:=0;  //default
mb_Input_Registers[164]:=0;  //default
mb_Input_Registers[165]:=0;  //default
mb_Input_Registers[166]:=0;  //default
mb_Input_Registers[167]:=0;  //default
mb_Input_Registers[168]:=0;  //default
mb_Input_Registers[169]:=0;  //default
mb_Input_Registers[170]:=0;  //default
mb_Input_Registers[171]:=0;  //default
mb_Input_Registers[172]:=0;  //default
mb_Input_Registers[173]:=0;  //default
mb_Input_Registers[174]:=0;  //default
mb_Input_Registers[175]:=0;  //default
mb_Input_Registers[176]:=0;  //default
mb_Input_Registers[177]:=0;  //default
mb_Input_Registers[178]:=0;  //default
mb_Input_Registers[179]:=0;  //default
mb_Input_Registers[180]:=0;  //default
mb_Input_Registers[181]:=0;  //default
mb_Input_Registers[182]:=0;  //default
mb_Input_Registers[183]:=0;  //default
mb_Input_Registers[184]:=0;  //default
mb_Input_Registers[185]:=0;  //default
mb_Input_Registers[186]:=0;  //default
mb_Input_Registers[187]:=0;  //default
mb_Input_Registers[188]:=0;  //default
mb_Input_Registers[189]:=0;  //default
mb_Input_Registers[190]:=0;  //default
mb_Input_Registers[191]:=0;  //default
mb_Input_Registers[192]:=0;  //default
mb_Input_Registers[193]:=0;  //default
mb_Input_Registers[194]:=0;  //default
mb_Input_Registers[195]:=0;  //default
mb_Input_Registers[196]:=0;  //default
mb_Input_Registers[197]:=0;  //default
mb_Input_Registers[198]:=0;  //default
mb_Input_Registers[199]:=0;  //default
mb_Input_Registers[200]:=0;  //default
mb_Input_Registers[201]:=0;  //default
mb_Input_Registers[202]:=0;  //default
mb_Input_Registers[203]:=0;  //default
mb_Input_Registers[204]:=0;  //default
mb_Input_Registers[205]:=0;  //default
mb_Input_Registers[206]:=0;  //default
mb_Input_Registers[207]:=0;  //default
mb_Input_Registers[208]:=0;  //default
mb_Input_Registers[209]:=0;  //default
mb_Input_Registers[210]:=0;  //default
mb_Input_Registers[211]:=0;  //default
mb_Input_Registers[212]:=0;  //default
mb_Input_Registers[213]:=0;  //default
mb_Input_Registers[214]:=0;  //default
mb_Input_Registers[215]:=0;  //default
mb_Input_Registers[216]:=0;  //default
mb_Input_Registers[217]:=0;  //default
mb_Input_Registers[218]:=0;  //default
mb_Input_Registers[219]:=0;  //default
mb_Input_Registers[220]:=0;  //default
mb_Input_Registers[221]:=0;  //default
mb_Input_Registers[222]:=0;  //default
mb_Input_Registers[223]:=0;  //default
mb_Input_Registers[224]:=0;  //default
mb_Input_Registers[225]:=0;  //default
mb_Input_Registers[226]:=0;  //default
mb_Input_Registers[227]:=0;  //default
mb_Input_Registers[228]:=0;  //default
mb_Input_Registers[229]:=0;  //default
mb_Input_Registers[230]:=0;  //default
mb_Input_Registers[231]:=0;  //default
mb_Input_Registers[232]:=0;  //default
mb_Input_Registers[233]:=0;  //default
mb_Input_Registers[234]:=0;  //default
mb_Input_Registers[235]:=0;  //default
mb_Input_Registers[236]:=0;  //default
mb_Input_Registers[237]:=0;  //default
mb_Input_Registers[238]:=0;  //default
mb_Input_Registers[239]:=0;  //default
mb_Input_Registers[240]:=0;  //default
mb_Input_Registers[241]:=0;  //default
mb_Input_Registers[242]:=0;  //default
mb_Input_Registers[243]:=0;  //default
mb_Input_Registers[244]:=0;  //default
mb_Input_Registers[245]:=0;  //default
mb_Input_Registers[246]:=0;  //default
mb_Input_Registers[247]:=0;  //default
mb_Input_Registers[248]:=0;  //default
mb_Input_Registers[249]:=0;  //default
mb_Input_Registers[250]:=0;  //default
mb_Input_Registers[251]:=0;  //default
mb_Input_Registers[252]:=0;  //default
mb_Input_Registers[253]:=0;  //default
mb_Input_Registers[254]:=0;  //default
mb_Input_Registers[255]:=0;  //default

END_PROGRAM

// ---- POUs/Modbus/p_ModbusTx_PLCMemory.TcPOU
PROGRAM p_ModbusTx_PLCMemory
VAR

END_VAR

MEMCPY(srcAddr:=ADR(HOMS2_XGantry.PAxis.stStatus.rActPosition), destAddr:=ADR(mb_PLC_Memory[130]), n:=SIZEOF(HOMS2_XGantry.PAxis.stStatus.rActPosition));
MEMCPY(srcAddr:=ADR(HOMS2_XGantry.PAxis.stStatus.rActVelocity), destAddr:=ADR(mb_PLC_Memory[132]), n:=SIZEOF(HOMS2_XGantry.PAxis.stStatus.rActVelocity));
MEMCPY(srcAddr:=ADR(HOMS2_XGantry.PAxis.stAxis.NcToPlc.SetAcc), destAddr:=ADR(mb_PLC_Memory[134]), n:=SIZEOF(HOMS2_XGantry.PAxis.stAxis.NcToPlc.SetAcc));
MEMCPY(srcAddr:=ADR(HOMS2_XGantry.SAxis.stStatus.rActPosition), destAddr:=ADR(mb_PLC_Memory[136]), n:=SIZEOF(HOMS2_XGantry.SAxis.stStatus.rActPosition));
MEMCPY(srcAddr:=ADR(HOMS2_XGantry.SAxis.stStatus.rActVelocity), destAddr:=ADR(mb_PLC_Memory[138]), n:=SIZEOF(HOMS2_XGantry.SAxis.stStatus.rActVelocity));
MEMCPY(srcAddr:=ADR(HOMS2_XGantry.SAxis.stAxis.NcToPlc.SetAcc), destAddr:=ADR(mb_PLC_Memory[140]), n:=SIZEOF(HOMS2_XGantry.SAxis.stAxis.NcToPlc.SetAcc));
MEMCPY(srcAddr:=ADR(HOMS2_YGantry.PAxis.stStatus.rActPosition), destAddr:=ADR(mb_PLC_Memory[142]), n:=SIZEOF(HOMS2_YGantry.PAxis.stStatus.rActPosition));
MEMCPY(srcAddr:=ADR(HOMS2_YGantry.PAxis.stStatus.rActVelocity), destAddr:=ADR(mb_PLC_Memory[144]), n:=SIZEOF(HOMS2_YGantry.PAxis.stStatus.rActVelocity));
MEMCPY(srcAddr:=ADR(HOMS2_YGantry.PAxis.stAxis.NcToPlc.SetAcc), destAddr:=ADR(mb_PLC_Memory[146]), n:=SIZEOF(HOMS2_YGantry.PAxis.stAxis.NcToPlc.SetAcc));
MEMCPY(srcAddr:=ADR(HOMS2_YGantry.SAxis.stStatus.rActPosition), destAddr:=ADR(mb_PLC_Memory[148]), n:=SIZEOF(HOMS2_YGantry.SAxis.stStatus.rActPosition));
MEMCPY(srcAddr:=ADR(HOMS2_YGantry.SAxis.stStatus.rActVelocity), destAddr:=ADR(mb_PLC_Memory[150]), n:=SIZEOF(HOMS2_YGantry.SAxis.stStatus.rActVelocity));
MEMCPY(srcAddr:=ADR(HOMS2_YGantry.SAxis.stAxis.NcToPlc.SetAcc), destAddr:=ADR(mb_PLC_Memory[152]), n:=SIZEOF(HOMS2_YGantry.SAxis.stAxis.NcToPlc.SetAcc));
MEMCPY(srcAddr:=ADR(HOMS2_Pitch.Stepper.stStatus.rActPosition), destAddr:=ADR(mb_PLC_Memory[154]), n:=SIZEOF(HOMS2_Pitch.Stepper.stStatus.rActPosition));
MEMCPY(srcAddr:=ADR(HOMS2_Pitch.Stepper.stStatus.rActVelocity), destAddr:=ADR(mb_PLC_Memory[156]), n:=SIZEOF(HOMS2_Pitch.Stepper.stStatus.rActVelocity));
MEMCPY(srcAddr:=ADR(HOMS2_Pitch.Stepper.stAxis.NcToPlc.SetAcc), destAddr:=ADR(mb_PLC_Memory[158]), n:=SIZEOF(HOMS2_Pitch.Stepper.stAxis.NcToPlc.SetAcc));

MEMCPY(srcAddr:=ADR(HOMS2_Pitch.Piezo.rActVoltage), destAddr:=ADR(mb_PLC_Memory[166]), n:=SIZEOF(HOMS2_Pitch.Piezo.rActVoltage));
MEMCPY(srcAddr:=ADR(HOMS2_Pitch.Piezo.UpperVoltage), destAddr:=ADR(mb_PLC_Memory[168]), n:=SIZEOF(HOMS2_Pitch.Piezo.UpperVoltage));
MEMCPY(srcAddr:=ADR(HOMS2_Pitch.Piezo.LowerVoltage), destAddr:=ADR(mb_PLC_Memory[170]), n:=SIZEOF(HOMS2_Pitch.Piezo.LowerVoltage));

MEMCPY(srcAddr:=ADR(HOMS2_XGantry.DiffTol), destAddr:=ADR(mb_PLC_Memory[180]), n:=SIZEOF(HOMS2_XGantry.DiffTol));
MEMCPY(srcAddr:=ADR(HOMS2_XGantry.Diff), destAddr:=ADR(mb_PLC_Memory[182]), n:=SIZEOF(HOMS2_XGantry.Diff));
MEMCPY(srcAddr:=ADR(HOMS2_YGantry.DiffTol), destAddr:=ADR(mb_PLC_Memory[184]), n:=SIZEOF(HOMS2_YGantry.DiffTol));
MEMCPY(srcAddr:=ADR(HOMS2_YGantry.Diff), destAddr:=ADR(mb_PLC_Memory[186]), n:=SIZEOF(HOMS2_YGantry.Diff));




MEMCPY(destAddr:=ADR(mb_PLC_Memory[36]), srcAddr:=ADR(HOMS2_Pitch.Axis.rReqAbsPos), n:=SIZEOF(HOMS2_Pitch.Axis.rReqAbsPos));
MEMCPY(destAddr:=ADR(mb_PLC_Memory[56]), srcAddr:=ADR(HOMS3_Pitch.Axis.rReqAbsPos), n:=SIZEOF(HOMS3_Pitch.Axis.rReqAbsPos));

MEMCPY(srcAddr:=ADR(HOMS3_XGantry.PAxis.stStatus.rActPosition), destAddr:=ADR(mb_PLC_Memory[188]), n:=SIZEOF(HOMS3_XGantry.PAxis.stStatus.rActPosition));
MEMCPY(srcAddr:=ADR(HOMS3_XGantry.PAxis.stStatus.rActVelocity), destAddr:=ADR(mb_PLC_Memory[190]), n:=SIZEOF(HOMS3_XGantry.PAxis.stStatus.rActVelocity));
MEMCPY(srcAddr:=ADR(HOMS3_XGantry.PAxis.stAxis.NcToPlc.SetAcc), destAddr:=ADR(mb_PLC_Memory[192]), n:=SIZEOF(HOMS3_XGantry.PAxis.stAxis.NcToPlc.SetAcc));
MEMCPY(srcAddr:=ADR(HOMS3_XGantry.SAxis.stStatus.rActPosition), destAddr:=ADR(mb_PLC_Memory[194]), n:=SIZEOF(HOMS3_XGantry.SAxis.stStatus.rActPosition));
MEMCPY(srcAddr:=ADR(HOMS3_XGantry.SAxis.stStatus.rActVelocity), destAddr:=ADR(mb_PLC_Memory[196]), n:=SIZEOF(HOMS3_XGantry.SAxis.stStatus.rActVelocity));
MEMCPY(srcAddr:=ADR(HOMS3_XGantry.SAxis.stAxis.NcToPlc.SetAcc), destAddr:=ADR(mb_PLC_Memory[198]), n:=SIZEOF(HOMS3_XGantry.SAxis.stAxis.NcToPlc.SetAcc));
MEMCPY(srcAddr:=ADR(HOMS3_YGantry.PAxis.stStatus.rActPosition), destAddr:=ADR(mb_PLC_Memory[200]), n:=SIZEOF(HOMS3_YGantry.PAxis.stStatus.rActPosition));
MEMCPY(srcAddr:=ADR(HOMS3_YGantry.PAxis.stStatus.rActVelocity), destAddr:=ADR(mb_PLC_Memory[202]), n:=SIZEOF(HOMS3_YGantry.PAxis.stStatus.rActVelocity));
MEMCPY(srcAddr:=ADR(HOMS3_YGantry.PAxis.stAxis.NcToPlc.SetAcc), destAddr:=ADR(mb_PLC_Memory[204]), n:=SIZEOF(HOMS3_YGantry.PAxis.stAxis.NcToPlc.SetAcc));
MEMCPY(srcAddr:=ADR(HOMS3_YGantry.SAxis.stStatus.rActPosition), destAddr:=ADR(mb_PLC_Memory[206]), n:=SIZEOF(HOMS3_YGantry.SAxis.stStatus.rActPosition));
MEMCPY(srcAddr:=ADR(HOMS3_YGantry.SAxis.stStatus.rActVelocity), destAddr:=ADR(mb_PLC_Memory[208]), n:=SIZEOF(HOMS3_YGantry.SAxis.stStatus.rActVelocity));
MEMCPY(srcAddr:=ADR(HOMS3_YGantry.SAxis.stAxis.NcToPlc.SetAcc), destAddr:=ADR(mb_PLC_Memory[210]), n:=SIZEOF(HOMS3_YGantry.SAxis.stAxis.NcToPlc.SetAcc));
MEMCPY(srcAddr:=ADR(HOMS3_Pitch.Stepper.stStatus.rActPosition), destAddr:=ADR(mb_PLC_Memory[212]), n:=SIZEOF(HOMS3_Pitch.Stepper.stStatus.rActPosition));
MEMCPY(srcAddr:=ADR(HOMS3_Pitch.Stepper.stStatus.rActVelocity), destAddr:=ADR(mb_PLC_Memory[214]), n:=SIZEOF(HOMS3_Pitch.Stepper.stStatus.rActVelocity));
MEMCPY(srcAddr:=ADR(HOMS3_Pitch.Stepper.stAxis.NcToPlc.SetAcc), destAddr:=ADR(mb_PLC_Memory[216]), n:=SIZEOF(HOMS3_Pitch.Stepper.stAxis.NcToPlc.SetAcc));
MEMCPY(srcAddr:=ADR(HOMS3_Pitch.Piezo.rActVoltage), destAddr:=ADR(mb_PLC_Memory[218]), n:=SIZEOF(HOMS3_Pitch.Piezo.rActVoltage));
MEMCPY(srcAddr:=ADR(HOMS3_Pitch.Piezo.UpperVoltage), destAddr:=ADR(mb_PLC_Memory[220]), n:=SIZEOF(HOMS3_Pitch.Piezo.UpperVoltage));
MEMCPY(srcAddr:=ADR(HOMS3_Pitch.Piezo.LowerVoltage), destAddr:=ADR(mb_PLC_Memory[222]), n:=SIZEOF(HOMS3_Pitch.Piezo.LowerVoltage));
MEMCPY(srcAddr:=ADR(HOMS3_XGantry.DiffTol), destAddr:=ADR(mb_PLC_Memory[224]), n:=SIZEOF(HOMS3_XGantry.DiffTol));
MEMCPY(srcAddr:=ADR(HOMS3_XGantry.Diff), destAddr:=ADR(mb_PLC_Memory[226]), n:=SIZEOF(HOMS3_XGantry.Diff));
MEMCPY(srcAddr:=ADR(HOMS3_YGantry.DiffTol), destAddr:=ADR(mb_PLC_Memory[228]), n:=SIZEOF(HOMS3_YGantry.DiffTol));
MEMCPY(srcAddr:=ADR(HOMS3_YGantry.Diff), destAddr:=ADR(mb_PLC_Memory[230]), n:=SIZEOF(HOMS3_YGantry.Diff));


MEMCPY(srcAddr:=ADR(HOMS2_Pitch.ReqPosLimLo), destAddr:=ADR(mb_PLC_Memory[236]), n:=SIZEOF(HOMS2_Pitch.ReqPosLimLo));
MEMCPY(srcAddr:=ADR(HOMS2_Pitch.ReqPosLimHi), destAddr:=ADR(mb_PLC_Memory[238]), n:=SIZEOF(HOMS2_Pitch.ReqPosLimHi));
MEMCPY(srcAddr:=ADR(HOMS3_Pitch.ReqPosLimLo), destAddr:=ADR(mb_PLC_Memory[240]), n:=SIZEOF(HOMS3_Pitch.ReqPosLimLo));
MEMCPY(srcAddr:=ADR(HOMS3_Pitch.ReqPosLimHi), destAddr:=ADR(mb_PLC_Memory[242]), n:=SIZEOF(HOMS3_Pitch.ReqPosLimHi));


MEMCPY(destAddr:=ADR(mb_PLC_Memory[64]), srcAddr:=ADR(HOMS2_Pitch.Stepper.rStepperDmovRange), n:=SIZEOF(HOMS2_Pitch.Stepper.rStepperDmovRange));
MEMCPY(destAddr:=ADR(mb_PLC_Memory[66]), srcAddr:=ADR(HOMS2_Pitch.Piezo.rPiezoDmovRange), n:=SIZEOF(HOMS2_Pitch.Piezo.rPiezoDmovRange));
MEMCPY(destAddr:=ADR(mb_PLC_Memory[68]), srcAddr:=ADR(HOMS3_Pitch.Stepper.rStepperDmovRange), n:=SIZEOF(HOMS3_Pitch.Stepper.rStepperDmovRange));
MEMCPY(destAddr:=ADR(mb_PLC_Memory[70]), srcAddr:=ADR(HOMS3_Pitch.Piezo.rPiezoDmovRange), n:=SIZEOF(HOMS3_Pitch.Piezo.rPiezoDmovRange));


//MEMCPY(destAddr:=ADR(mb_PLC_Memory[256]), srcAddr:=ADR(HOMS3_Pitch.Axis.rReqAbsPos), n:=SIZEOF(HOMS3_Pitch.Stepper.rReqAbsolute));

END_PROGRAM

// ---- POUs/Modbus/p_ModbusTx_OutputCoils.TcPOU
PROGRAM p_ModbusTx_OutputCoils
VAR

END_VAR

mb_Output_Coils[0]:=FALSE;  //System Controls
mb_Output_Coils[1]:=g_stSystem.xOverrideMode;  //System Controls
mb_Output_Coils[2]:=q_xDG1_MMS01_MPSOK ;  //System Controls
mb_Output_Coils[3] :=q_xMFX_VGC_OK;  //System Controls
mb_Output_Coils[4] :=q_xMFX_preS45_MPSOK;  //System Controls
mb_Output_Coils[5] :=q_xMFX_MPSOK;  //System Controlsmb_Output_Coils[2]:=FALSE;  //System Controls
mb_Output_Coils[6]:=FALSE;  //System Controls
mb_Output_Coils[7]:=FALSE;  //System Controls
mb_Output_Coils[8]:=FALSE;  //System Controls
mb_Output_Coils[9]:=FALSE;  //System Controls
mb_Output_Coils[10]:=vgcMXT_VGC_04.xOPN_SW;  //Valve switch controls
mb_Output_Coils[11]:=vgcDVD_VGC_01.xOPN_SW;  //Valve switch controls
mb_Output_Coils[12]:=vgcDIA_VGC_01.xOPN_SW;  //Valve switch controls
mb_Output_Coils[13]:=vgcDIA_VGC_02.xOPN_SW;  //Valve switch controls
mb_Output_Coils[14]:=vgcDG1_VGC_01.xOPN_SW;  //Valve switch controls
mb_Output_Coils[15]:=vgcDG1_VGC_02.xOPN_SW;  //Valve switch controls
mb_Output_Coils[16]:=FALSE;  //Valve switch controls
mb_Output_Coils[17]:=FALSE;  //Valve switch controls
mb_Output_Coils[18]:=FALSE;  //Valve switch controls
mb_Output_Coils[19]:=FALSE;  //Valve switch controls
mb_Output_Coils[20]:=FALSE;  //Valve switch controls
mb_Output_Coils[21]:=FALSE;  //Valve switch controls
mb_Output_Coils[22]:=FALSE;  //Valve switch controls
mb_Output_Coils[23]:=FALSE;  //Valve switch controls
mb_Output_Coils[24]:=FALSE;  //Valve switch controls
mb_Output_Coils[25]:=FALSE;  //Valve switch controls
mb_Output_Coils[26]:=FALSE;  //Valve switch controls
mb_Output_Coils[27]:=FALSE;  //Valve switch controls
mb_Output_Coils[28]:=FALSE;  //Valve switch controls
mb_Output_Coils[29]:=FALSE;  //Valve switch controls
mb_Output_Coils[30]:=FALSE;  //Valve switch controls
mb_Output_Coils[31]:=FALSE;  //Valve switch controls
mb_Output_Coils[32]:=FALSE;  //Valve switch controls
mb_Output_Coils[33]:=FALSE;  //Valve switch controls
mb_Output_Coils[34]:=FALSE;  //Valve switch controls
mb_Output_Coils[35]:=FALSE;  //Valve switch controls
mb_Output_Coils[36]:=FALSE;  //Valve switch controls
mb_Output_Coils[37]:=FALSE;  //Valve switch controls
mb_Output_Coils[38]:=FALSE;  //Valve switch controls
mb_Output_Coils[39]:=FALSE;  //Valve switch controls
mb_Output_Coils[40]:=FALSE;  //Valve switch controls
mb_Output_Coils[41]:=FALSE;  //Valve switch controls
mb_Output_Coils[42]:=FALSE;  //Valve switch controls
mb_Output_Coils[43]:=FALSE;  //Valve switch controls
mb_Output_Coils[44]:=FALSE;  //Valve switch controls
mb_Output_Coils[45]:=FALSE;  //Valve switch controls
mb_Output_Coils[46]:=FALSE;  //Valve switch controls
mb_Output_Coils[47]:=FALSE;  //Valve switch controls
mb_Output_Coils[48]:=FALSE;  //Valve switch controls
mb_Output_Coils[49]:=FALSE;  //Valve switch controls
mb_Output_Coils[50]:=FALSE;  //Valve switch controls
mb_Output_Coils[51]:=FALSE;  //Valve switch controls
mb_Output_Coils[52]:=FALSE;  //Valve switch controls
mb_Output_Coils[53]:=FALSE;  //Valve switch controls
mb_Output_Coils[54]:=FALSE;  //Valve switch controls
mb_Output_Coils[55]:=FALSE;  //Valve switch controls
mb_Output_Coils[56]:=FALSE;  //Valve switch controls
mb_Output_Coils[57]:=FALSE;  //Valve switch controls
mb_Output_Coils[58]:=FALSE;  //Valve switch controls
mb_Output_Coils[59]:=FALSE;  //Valve switch controls
mb_Output_Coils[60]:=FALSE;  //Valve switch controls
mb_Output_Coils[61]:=FALSE;  //Valve switch controls
mb_Output_Coils[62]:=FALSE;  //Valve switch controls
mb_Output_Coils[63]:=FALSE;  //Valve switch controls
mb_Output_Coils[64]:=FALSE;  //Valve switch controls
mb_Output_Coils[65]:=FALSE;  //Valve switch controls
mb_Output_Coils[66]:=FALSE;  //Valve switch controls
mb_Output_Coils[67]:=FALSE;  //Valve switch controls
mb_Output_Coils[68]:=FALSE;  //Valve switch controls
mb_Output_Coils[69]:=FALSE;  //Valve switch controls
mb_Output_Coils[70]:=FALSE;  //Turbo Controls
mb_Output_Coils[71]:=FALSE;  //Turbo Controls
mb_Output_Coils[72]:=FALSE;  //Turbo Controls
mb_Output_Coils[74]:=FALSE;  //Turbo Controls
mb_Output_Coils[75]:=FALSE;  //Turbo Controls
mb_Output_Coils[76]:=FALSE;  //Turbo Controls
mb_Output_Coils[77]:=FALSE;  //Turbo Controls
mb_Output_Coils[78]:=FALSE;  //Turbo Controls
mb_Output_Coils[79]:=FALSE;  //Turbo Controls
mb_Output_Coils[80]:=FALSE;  //Turbo Controls
mb_Output_Coils[81]:=FALSE;  //Turbo Controls
mb_Output_Coils[82]:=FALSE;  //Turbo Controls
mb_Output_Coils[83]:=FALSE;  //Turbo Controls
mb_Output_Coils[84]:=FALSE;  //Turbo Controls
mb_Output_Coils[85]:=FALSE;  //Turbo Controls
mb_Output_Coils[86]:=FALSE;  //Turbo Controls
mb_Output_Coils[87]:=FALSE;  //Turbo Controls
mb_Output_Coils[88]:=FALSE;  //Turbo Controls
mb_Output_Coils[89]:=FALSE;  //Turbo Controls
mb_Output_Coils[90]:=FALSE;  //Turbo Controls
mb_Output_Coils[91]:=FALSE;  //Turbo Controls
mb_Output_Coils[92]:=FALSE;  //Turbo Controls
mb_Output_Coils[93]:=FALSE;  //Turbo Controls
mb_Output_Coils[94]:=FALSE;  //Turbo Controls
mb_Output_Coils[95]:=FALSE;  //Turbo Controls
mb_Output_Coils[96]:=FALSE;  //Turbo Controls
mb_Output_Coils[97]:=FALSE;  //Turbo Controls
mb_Output_Coils[98]:=FALSE;  //Turbo Controls
mb_Output_Coils[99]:=FALSE;  //Turbo Controls
mb_Output_Coils[100]:=FALSE;  //Turbo Controls
mb_Output_Coils[101]:=FALSE;  //Turbo Controls
mb_Output_Coils[102]:=FALSE;  //Turbo Controls
mb_Output_Coils[103]:=FALSE;  //Turbo Controls
mb_Output_Coils[104]:=FALSE;  //Turbo Controls
mb_Output_Coils[105]:=FALSE;  //Turbo Controls
mb_Output_Coils[106]:=FALSE;  //Turbo Controls
mb_Output_Coils[107]:=FALSE;  //Turbo Controls
mb_Output_Coils[108]:=FALSE;  //Turbo Controls
mb_Output_Coils[109]:=FALSE;  //Turbo Controls
mb_Output_Coils[110]:=FALSE;  //Turbo Controls
mb_Output_Coils[111]:=FALSE;  //Turbo Controls
mb_Output_Coils[112]:=FALSE;  //Turbo Controls
mb_Output_Coils[113]:=FALSE;  //Turbo Controls
mb_Output_Coils[114]:=FALSE;  //Turbo Controls
mb_Output_Coils[115]:=FALSE;  //Turbo Controls
mb_Output_Coils[116]:=FALSE;  //Turbo Controls
mb_Output_Coils[117]:=FALSE;  //Turbo Controls
mb_Output_Coils[118]:=FALSE;  //Turbo Controls
mb_Output_Coils[119]:=FALSE;  //Turbo Controls
//mb_Output_Coils[120]:=vgMXT_GCC_06.xHV_SW;  //CC HV Enable
mb_Output_Coils[121]:=vgDVD_GCC_02.xHV_SW;  //CC HV Enable
mb_Output_Coils[122]:=vgDVD_GCC_04.xHV_SW;  //CC HV Enable
mb_Output_Coils[123]:=vgMON_GCC_01.xHV_SW;  //CC HV Enable
mb_Output_Coils[124]:=vgDIA_GCC_01.xHV_SW;  //CC HV Enable
mb_Output_Coils[125]:=vgSB2_GCC_01.xHV_SW;  //CC HV Enable
mb_Output_Coils[126]:=vgDG1_GCC_01.xHV_SW;  //CC HV Enable
mb_Output_Coils[127]:=vgDG2_GCC_01.xHV_SW;  //CC HV Enable
mb_Output_Coils[128]:=vgTFS_GCC_01.xHV_SW;  //CC HV Enable
mb_Output_Coils[129]:=FALSE;  //CC HV Enable
mb_Output_Coils[130]:=FALSE;  //CC HV Enable
mb_Output_Coils[131]:=FALSE;  //CC HV Enable
mb_Output_Coils[132]:=FALSE;  //CC HV Enable
mb_Output_Coils[133]:=FALSE;  //CC HV Enable
mb_Output_Coils[134]:=FALSE;  //CC HV Enable
mb_Output_Coils[135]:=FALSE;  //CC HV Enable
mb_Output_Coils[136]:=FALSE;  //CC HV Enable
mb_Output_Coils[137]:=FALSE;  //CC HV Enable
mb_Output_Coils[138]:=FALSE;  //CC HV Enable
mb_Output_Coils[139]:=FALSE;  //CC HV Enable
mb_Output_Coils[140]:=FALSE;  //CC HV Enable
mb_Output_Coils[141]:=FALSE;  //CC HV Enable
mb_Output_Coils[142]:=FALSE;  //CC HV Enable
mb_Output_Coils[143]:=FALSE;  //CC HV Enable
mb_Output_Coils[144]:=FALSE;  //CC HV Enable
mb_Output_Coils[145]:=FALSE;  //CC HV Enable
mb_Output_Coils[146]:=FALSE;  //CC HV Enable
mb_Output_Coils[147]:=FALSE;  //CC HV Enable
mb_Output_Coils[148]:=FALSE;  //CC HV Enable
mb_Output_Coils[149]:=FALSE;  //CC HV Enable
mb_Output_Coils[150]:=FALSE;  //CC HV Enable
mb_Output_Coils[151]:=FALSE;  //CC HV Enable
mb_Output_Coils[152]:=FALSE;  //CC HV Enable
mb_Output_Coils[153]:=FALSE;  //CC HV Enable
mb_Output_Coils[154]:=FALSE;  //CC HV Enable
mb_Output_Coils[155]:=FALSE;  //CC HV Enable
mb_Output_Coils[156]:=FALSE;  //CC HV Enable
mb_Output_Coils[157]:=FALSE;  //CC HV Enable
mb_Output_Coils[158]:=FALSE;  //CC HV Enable
mb_Output_Coils[159]:=FALSE;  //CC HV Enable
mb_Output_Coils[160]:=FALSE;  //
mb_Output_Coils[161]:=FALSE;  //
mb_Output_Coils[162]:=FALSE;  //
mb_Output_Coils[163]:=FALSE;  //
mb_Output_Coils[164]:=FALSE;  //
mb_Output_Coils[165]:=FALSE;  //
mb_Output_Coils[166]:=FALSE;  //
mb_Output_Coils[167]:=FALSE;  //
mb_Output_Coils[168]:=FALSE;  //
mb_Output_Coils[169]:=FALSE;  //
mb_Output_Coils[170]:=FALSE;  //
mb_Output_Coils[171]:=FALSE;  //
mb_Output_Coils[172]:=FALSE;  //
mb_Output_Coils[173]:=FALSE;  //
mb_Output_Coils[174]:=FALSE;  //
mb_Output_Coils[175]:=FALSE;  //
mb_Output_Coils[176]:=FALSE;  //
mb_Output_Coils[177]:=FALSE;  //
mb_Output_Coils[178]:=FALSE;  //
mb_Output_Coils[179]:=FALSE;  //
mb_Output_Coils[180]:=FALSE;  //
mb_Output_Coils[181]:=FALSE;  //
mb_Output_Coils[182]:=FALSE;  //
mb_Output_Coils[183]:=FALSE;  //
mb_Output_Coils[184]:=FALSE;  //
mb_Output_Coils[185]:=FALSE;  //
mb_Output_Coils[186]:=FALSE;  //
mb_Output_Coils[187]:=FALSE;  //
mb_Output_Coils[188]:=FALSE;  //
mb_Output_Coils[189]:=FALSE;  //
mb_Output_Coils[190]:=FALSE;  //
mb_Output_Coils[191]:=FALSE;  //
mb_Output_Coils[192]:=FALSE;  //
mb_Output_Coils[193]:=FALSE;  //
mb_Output_Coils[194]:=FALSE;  //
mb_Output_Coils[195]:=FALSE;  //
mb_Output_Coils[196]:=FALSE;  //
mb_Output_Coils[197]:=FALSE;  //
mb_Output_Coils[198]:=FALSE;  //
mb_Output_Coils[199]:=FALSE;  //
mb_Output_Coils[200]:=FALSE;  //Valve overrides
mb_Output_Coils[201]:=FALSE;  //Valve overrides
mb_Output_Coils[202]:=FALSE;  //Valve overrides
mb_Output_Coils[203]:=FALSE;  //Valve overrides
mb_Output_Coils[204]:=FALSE;  //
mb_Output_Coils[205]:=FALSE;  //
mb_Output_Coils[206]:=FALSE;  //
mb_Output_Coils[207]:=FALSE;  //
mb_Output_Coils[208]:=FALSE;  //
mb_Output_Coils[209]:=FALSE;  //
mb_Output_Coils[210]:=FALSE;  //
mb_Output_Coils[211]:=FALSE;  //
mb_Output_Coils[212]:=FALSE;  //
mb_Output_Coils[213]:=FALSE;  //
mb_Output_Coils[214]:=FALSE;  //
mb_Output_Coils[215]:=FALSE;  //
mb_Output_Coils[216]:=FALSE;  //
mb_Output_Coils[217]:=FALSE;  //
mb_Output_Coils[218]:=FALSE;  //
mb_Output_Coils[219]:=FALSE;  //
mb_Output_Coils[220]:=FALSE;  //
mb_Output_Coils[221]:=FALSE;  //
mb_Output_Coils[222]:=FALSE;  //
mb_Output_Coils[223]:=FALSE;  //
mb_Output_Coils[224]:=FALSE;  //
mb_Output_Coils[225]:=FALSE;  //
mb_Output_Coils[226]:=FALSE;  //
mb_Output_Coils[227]:=FALSE;  //
mb_Output_Coils[228]:=FALSE;  //
mb_Output_Coils[229]:=FALSE;  //
mb_Output_Coils[230]:=FALSE;  //
mb_Output_Coils[231]:=FALSE;  //
mb_Output_Coils[232]:=FALSE;  //
mb_Output_Coils[233]:=FALSE;  //
mb_Output_Coils[234]:=FALSE;  //
mb_Output_Coils[235]:=FALSE;  //
mb_Output_Coils[236]:=FALSE;  //
mb_Output_Coils[237]:=FALSE;  //
mb_Output_Coils[238]:=FALSE;  //
mb_Output_Coils[239]:=FALSE;  //
mb_Output_Coils[240]:=FALSE;  //
mb_Output_Coils[241]:=FALSE;  //
mb_Output_Coils[242]:=FALSE;  //
mb_Output_Coils[243]:=FALSE;  //
mb_Output_Coils[244]:=FALSE;  //
mb_Output_Coils[245]:=FALSE;  //
mb_Output_Coils[246]:=FALSE;  //
mb_Output_Coils[247]:=FALSE;  //
mb_Output_Coils[248]:=FALSE;  //
mb_Output_Coils[249]:=FALSE;  //
mb_Output_Coils[250]:=FALSE;  //
mb_Output_Coils[251]:=FALSE;  //
mb_Output_Coils[252]:=FALSE;  //
mb_Output_Coils[253]:=FALSE;  //
mb_Output_Coils[254]:=FALSE;  //
mb_Output_Coils[255]:=FALSE;  //

END_PROGRAM

// ---- POUs/Serial Comm/PiezoSerial.TcPOU
PROGRAM PiezoSerial
VAR
	//PI Serial
	fbE621SerialDriver_XRTM1 : FB_PI_E621_SerialDriver;
	rtInitParams_XRTM1	:	R_TRIG;
	tonTimeoutRst_XRTM1	: TON := (PT:=T#2S); //For timeout reset
	
	fbE621SerialDriverM2 : FB_PI_E621_SerialDriver;
	fbE621SerialDriverM3 : FB_PI_E621_SerialDriver;
	tonTimeoutRstM2	: TON := (PT:=T#2S); //For timeout reset
END_VAR

//Piezo E-621
///////////////////////
fbE621SerialDriver_XRTM1.i_xExecute := TRUE;
fbE621SerialDriver_XRTM1.i_xExecute R= fbE621SerialDriver_XRTM1.q_xDone;
fbE621SerialDriver_XRTM1(iq_stPiezoAxis:= GVL_XRTM1.XRTM1_Pitch.Piezo,
		                iq_stSerialRXBuffer:= Serial_RXBuffer_XRTM1,
		                iq_stSerialTXBuffer:= Serial_TXBuffer_XRTM1);
						
//M2 Piezo E-621
///////////////////////
	fbE621SerialDriverM2.i_xExecute := TRUE;
	fbE621SerialDriverM2.i_xExecute R= fbE621SerialDriverM2.q_xDone;
	fbE621SerialDriverM2(
		iq_stPiezoAxis:= HOMS2_Pitch.Piezo, 
		iq_stSerialRXBuffer:= Serial_P2_SerialRXBuffer, 
		iq_stSerialTXBuffer:= Serial_P2_SerialTXBuffer);
		
//M3 Piezo E-621
///////////////////////
	fbE621SerialDriverM3.i_xExecute := TRUE;
	fbE621SerialDriverM3.i_xExecute R= fbE621SerialDriverM3.q_xDone;
	fbE621SerialDriverM3(
		iq_stPiezoAxis:= HOMS3_Pitch.Piezo, 
		iq_stSerialRXBuffer:= Serial_P3_SerialRXBuffer, 
		iq_stSerialTXBuffer:= Serial_P3_SerialTXBuffer);

END_PROGRAM

// ---- POUs/Serial Comm/P_Serial_Com.TcPOU
PROGRAM P_Serial_Com
VAR
	fbSerialLineControl_EL6001_XRTM1: SerialLineControl; // XRTM1 Serial Comm Function Block
	
	// M2
	fbSerialLineControl_EL6001_P2: SerialLineControl;
	// M3
	fbSerialLineControl_EL6001_P3: SerialLineControl;

END_VAR

// These are the global IOs...don't forget to copy your data into them

(* EL6001 Serial port 0 com function *)
fbSerialLineControl_EL6001_XRTM1(Mode:= SERIALLINEMODE_EL6_22B,
						        pComIn:= ADR(Serial_stComIn_XRTM1),
						   	    pComOut:=ADR(Serial_stComOut_XRTM1),
						        SizeComIn:= SIZEOF(Serial_stComIn_XRTM1),
						        TxBuffer:= Serial_TXBuffer_XRTM1,
						        RxBuffer:= Serial_RXBuffer_XRTM1,
						        Error=>,
						        ErrorID=>);
								
fbSerialLineControl_EL6001_P2(
	Mode:= SERIALLINEMODE_EL6_22B (*SERIALLINEMODE_KL6_22B_STANDARD*),
	pComIn:= ADR(Serial_P2_stComIn),
	pComOut:=ADR(Serial_P2_stComOut) ,
	SizeComIn:= SIZEOF(Serial_P2_stComIn),
	TxBuffer:= Serial_P2_SerialTXBuffer,
	RxBuffer:= Serial_P2_SerialRXBuffer,
	Error=> ,
	ErrorID=> );
fbSerialLineControl_EL6001_P3(
	Mode:= SERIALLINEMODE_EL6_22B (*SERIALLINEMODE_KL6_22B_STANDARD*),
	pComIn:= ADR(Serial_P3_stComIn),
	pComOut:=ADR(Serial_P3_stComOut) ,
	SizeComIn:= SIZEOF(Serial_P3_stComIn),
	TxBuffer:= Serial_P3_SerialTXBuffer,
	RxBuffer:= Serial_P3_SerialRXBuffer,
	Error=> ,
	ErrorID=> );

END_PROGRAM
